PROGRAM PRG_TEST
VAR
	fbCalculatorTest : FB_Calculator_Test;
END_VAR

TcUnit.RUN();

END_PROGRAM

(* stored: Version 1.1.0.1, ProductVersion 3.1.4024.14
   POU PRG_TEST: Id {d55c3114-d863-49a3-bf23-c86fce701baf}, SpecialFunc None *)
